FUNCTION proj18_TupleStruct_3: BOOL
VAR_INPUT
    tuple: TupleStruct_3;
END_VAR


        proj18_TupleStruct_3 := tuple.field18;

END_FUNCTION

(* stored: ProductVersion 3.1.0.18, Version 1.1.0.1 *)
